Staubli VAL3: reset.pgx

program reset()
begin
  //putln(taskStatus("closeGripper"))
  if taskStatus("closeGripper")==1
    taskKill("closeGripper")
  endIf
  if taskStatus("moveBin")==1
    taskKill("moveBin")
  endIf
  if taskStatus("moveGate")==1
    taskKill("moveGate")
  endIf
  if taskStatus("moveHome")==1
    taskKill("moveHome")
  endIf
  if taskStatus("moveOffside")==1
    taskKill("moveOffside")
  endIf
  if taskStatus("moveZero")==1
    taskKill("moveZero")
  endIf
  if taskStatus("pickSample")==1
    taskKill("pickSample")
  endIf
  if taskStatus("releaseSample")==1
    taskKill("releaseSample")
  endIf
  if taskStatus("stopMotor")==1
    taskKill("stopMotor")
  endIf
  if taskStatus("restartMotor")==1
    taskKill("restartMotor")
  endIf
  stopMove()
  resetMotion()
end
